Staubli VAL3: OpenSingnal.pgx

program OpenSingnal()
begin
  //外设1
  IO:dOut["dOut4"]=true
end
